(* 
| :Description: This function block represents basic digital output and can be used for creating an instance of signle digital output device. 
| To control the output state use property "Value" 
*)
FUNCTION_BLOCK FB_DigitalOutput EXTENDS FB_DigitalDevice IMPLEMENTS  I_DigitalOutput
VAR
	bOut AT %Q*: BOOL; (* Current value of output*)
END_VAR
(*
Version history:

+-------------+------------+----------------+----------+------------------------------------------+
|Date         | Version    | created under  | Author   | Remark                                   |
+=============+============+================+==========+==========================================+
|2021-11      | 1.0.0.0    | V3.1.4024.22   | ADBO     | Function block created                   |
+-------------+------------+----------------+----------+------------------------------------------+
|2022-02      | 1.1.0.0    | V3.1.4024.22   | ADBO     | Changed to child of FB_DigitalDevice     |
+-------------+------------+----------------+----------+------------------------------------------+

*)

PROPERTY Out : BOOL
GET
Out := bOut;
END_GET
SET
bOut := Out;
END_SET
END_PROPERTY

END_FUNCTION_BLOCK

(* stored: Version 1.1.0.1, ProductVersion 3.1.4024.12
   POU FB_DigitalOutput: Id {e4607e00-17b3-420f-bcdb-87a21e0ebb22}, SpecialFunc None
   Folder Properties: Id {1939476e-a2bf-4246-8136-dc67b97f0d45}
   Folder Parameters: Id {8e523254-fbee-446f-a73e-71c7994dadab}
   Property Out: Id {b94d6fa3-7701-4ced-bb03-56a2c7137ea4}
   Get Get: Id {731e923d-a692-4e2c-bb67-9b4c39310b99}
   Set Set: Id {9b5ef51e-171f-48e0-a52d-c50ec7dd59d2} *)
